# EPICS substitutions: plcApp_IntLock/exampleApp/Db/userHost.substitutions
# Example substitutions file

file "db/dbExample1.db" {
    { user = "jiangboHost" }
}

file db/dbExample2.db {
    pattern { user, no, scan }
        { "jiangboHost", 1, "1 second" }
        { "jiangboHost", 2, "2 second" }
        { "jiangboHost", 3, "5 second" }
}
